SYSTEM Test ECC System
  (* Version 1.0, 2008-04-21, Goran Cengic, Chalmers *)
  DEVICE Test Device : DeviceType_not_used
    RESOURCE Test Resource : ResourceType_not_used
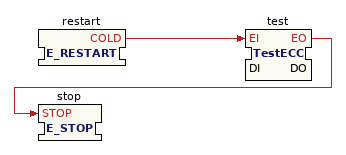
      FBS
        restart : E_RESTART;
        stop : E_STOP;
        test : TestECC;
      END_FBS
      EVENT_CONNECTIONS
        restart.COLD TO test.EI;
        test.EO TO stop.STOP;
      END_CONNECTIONS
    END_RESOURCE
  END_DEVICE
END_SYSTEM
